PROGRAM AquecimentoValvulas
VAR
	TON_Acionamento: TON;
	Iniciar	: BOOL;		//Inicia o aquecimento das válvulas
	Tempo	: DINT := 5;		//Tempo em que elas ficarão acionadas (s)
	VarAux: INT;
END_VAR
VAR_OUTPUT
	Acionar	:BOOL;
END_VAR

TON_Acionamento(IN:=Iniciar AND NOT TON_Acionamento.Q AND Testes.EmTeste, PT := DINT_TO_TIME(Tempo * 1000));

//Fica variando a variável auxiliar entre 0 e 1
IF TON_Acionamento.Q THEN
	IF VarAux = 0 THEN
		VarAux := 1;
	ELSE
		VarAux := 0;
	END_IF
END_IF

//Aciona a saída
Acionar := SEL(VarAux = 1, FALSE, TRUE);

END_PROGRAM

(* stored: Version 1.1.0.1, ProductVersion 3.1.4024.14
   POU AquecimentoValvulas: Id {19c3cf07-ea84-4369-9782-013a0ec287e3}, SpecialFunc None *)
